// TIA Portal V17 export
// export: Created 2025-06-26T06:33:58.2786582Z, ExportSetting WithDefaults, DisplayName Totally Integrated Automation Portal, DisplayVersion V17 Update 8, DisplayName TIA Portal Openness, DisplayVersion V17 Update 8, DisplayName TIA Portal Version Control Interface, DisplayVersion V17, DisplayName STEP 7 Professional, DisplayVersion V17 Update 8, DisplayName STEP 7 Safety, DisplayVersion V17 Update 6, DisplayName WinCC Advanced, DisplayVersion V17 Update 8
DATA_BLOCK "DB_DO"   // DB8
{ S7_Optimized_Access := 'TRUE' }
VERSION : 0.1
// stored: AutoNumber false, DBAccessibleFromOPCUA true, IsOnlyStoredInLoadMemory false, IsRetainMemResEnabled false, IsWriteProtectedInAS false, MemoryReserve 100
   VAR
      HBL_EC_01 : Bool;
      HBL_EC_02 : Bool;
      HBL_HV_630 : Bool;
      HBL_HV_114 : Bool;
      HBL_HV_115 : Bool;
      HBL_HV_860 : Bool;
      HBL_HV_861 : Bool;
      HBL_XV_06 : Bool;
      HBL_XV_07 : Bool;
      HBL_HV_631 : Bool;
      SSC_P_01 : Bool;
      SSC_F_01 : Bool;
      SSC_P_02 : Bool;
      CPC_P_01 : Bool;
      GH117_827 : Bool;   // Blowdown valve
      GH117_826_1 : Bool;   // NCG valve 1
      GH117_826_2 : Bool;   // NCG valve 2
      HBL_LSH_62 : Bool;
      HBL_LSL_63 : Bool;
      HBL_LSH_64 : Bool;
      HBL_LSL_864 : Bool;
      HBL_LS_632 : Bool;
      HBL_LS_633 : Bool;
   END_VAR
BEGIN
END_DATA_BLOCK
